(* CODESYS project SPT_Utilities.library
   Version: 4.0.1
   Title: SPT Utilities
   DefaultNamespace: SPT_Utilities
   Placeholder: SPT Utilities
   Company: Beckhoff Automation LLC

Project tree, tasks and I/O mapping:
  libraries: SPT Base Types, * (Beckhoff Automation LLC); SPT Event Logger, * (Beckhoff Automation LLC); Tc2_Standard, * (Beckhoff Automation GmbH); Tc2_System, * (Beckhoff Automation GmbH); Tc3_EventLogger, * (Beckhoff Automation GmbH); Tc3_JsonXml, * (Beckhoff Automation GmbH); Tc3_Module, * (Beckhoff Automation GmbH)
  Analog Scaling/
    DUT/
      data type ST_ScalingParameters
    function F_ApplyScaling [ST]
  Buffers/
    Array ANY Datatype/
      function block FB_ArrayAny [ST]: CheckBoundary, Delete, Enable, Exchange, Insert, LowerBoundary, Reset, UpperBoundary
    Buffers ANY Datatype/
      function block FB_AnyBase [ST]: CheckBoundary, CheckDataSize, CheckPointer, ClearError, Empty, Enable, Full, LowerBoundary, UpperBoundary
      function block FB_BufferAny [ST]: Push, Reset
      function block FB_FIFOAny [ST]: Pop, Push, Reset
      function block FB_LIFOAny [ST]: Pop, Push, Reset
      function block FB_RingAny [ST]: Pop, Push, Reset
      function IncrementBy1ToLimit [ST]
    function block FB_FIFO_ULINT_Array [ST]: AddEntry, EntryCount, LastInValue, NextOutValue, RemoveEntry
  File Handlers/
    function block FB_Component_JsonFileHandler [ST]: GetDataTypeFromPVOID, CreateEvents, Monitoring, CyclicLogic, ClearDocument, LoadFile, ReadAny, ReadBool, ReadDInt, ReadLREAL, ReadString, ReadSymbol, Reset, UpdateAny, UpdateBool, UpdateDInt, UpdateLREAL, UpdateString, UpdateSymbol, LoadFileSequence, SaveFileSequence, Path, Timeout
    interface I_FileHandler: ClearDocument, LoadFile, ReadBool, ReadDInt, ReadLREAL, ReadString, ReadSymbol, Reset, Timeout, UpdateAny, UpdateBool, UpdateDInt, UpdateLREAL, UpdateString, UpdateSymbol
  Helper/
    function F_CompareLREAL [ST]
    function F_CompareREAL [ST]
    function F_LREAL_RoundToPlace [ST]
    function block FB_SimpleRateLimiter [ST]
  Project Information/
    function F_GetCompany [ST]
    function F_GetTitle [ST]
    function F_GetVersion [ST]
  String Helper/
    function block FB_StringHelper [ST]: GetExtensionOrVarName, GetFileNameFromPath, GetFilePath, GetName, GetPath, GetSymbolPath, RemoveFirstChar, RemoveLastChar, StringToCharArray, ValidInput
  Trace Listener/
    function block FB_MessageListener [ST]: Listener, OnMessageSent
    function block FB_TraceListenerBase [ST]: CyclicLogic, Initialize, OnTraceReceived
    interface I_TraceListener: OnTraceReceived
    data type ST_TraceMessage
  Tree_IndexBased/
    function block FB_Tree_IndexBased [ST]: AddNodeAsChildByName, GetIndexByName, Initialize
    interface I_Tree_IndexBased: AddNodeAsChildByName
    data type ST_Tree_IndexBased_Node
  Version/
    global variables Global_Version
  00000000-0000-0000-0000-000000000000|LICENSE
  LICENSE
  global variables Parameter_Utilities
*)

// Analog Scaling/DUT/ST_ScalingParameters
TYPE ST_ScalingParameters :
	STRUCT
		Input_Minimum  : LREAL := 0;
		Input_Maximum  : LREAL := 100;
		Output_Minimum : LREAL := 0;
		Output_Maximum : LREAL := 4096;
	END_STRUCT
END_TYPE

// Trace Listener/ST_TraceMessage
TYPE ST_TraceMessage :
	STRUCT
		Timestamp : T_MaxString;
		Source	  : T_MaxString;
		Context	  : T_MaxString;
		ScanCount : UDINT;
		Flags	  : UDINT;
		Message	  : T_MaxString;
		Json	  : T_MaxString;
	END_STRUCT
END_TYPE

// Tree_IndexBased/ST_Tree_IndexBased_Node
TYPE ST_Tree_IndexBased_Node :
	STRUCT
		Name	   : STRING;
		ChildCount : DINT;
		Parent	   : DINT;
		Children   : ARRAY[0..15] OF DINT;
		Depth	   : DINT;
	END_STRUCT
END_TYPE

// Version/Global_Version
{attribute 'TcGenerated'}
{attribute 'no-analysis'}
{attribute 'linkalways'}
// This function has been automatically generated from the project information.
VAR_GLOBAL CONSTANT
	{attribute 'const_non_replaced'}
	stLibVersion_SPT_Utilities : ST_LibVersion := (iMajor := 4, iMinor := 0, iBuild := 1, iRevision := 0, nFlags := 1, sVersion := '4.0.1');
END_VAR

// Parameter_Utilities
{attribute 'qualified_only'}
VAR_GLOBAL CONSTANT
	FILE_SIZE : UDINT := 1300000; // Number of Characters in file to read via Read/Write Symbol
END_VAR

// Analog Scaling/F_ApplyScaling
FUNCTION F_ApplyScaling : LREAL
VAR_INPUT
	X		   : LREAL;
	Parameters : ST_ScalingParameters;
END_VAR

VAR
	Slope : LREAL;
END_VAR

IF Parameters.Input_Minimum >= Parameters.Input_Maximum THEN
	// Error -- no span to scale
	F_ApplyScaling := 0;
	RETURN;
ELSIF Parameters.Output_Minimum >= Parameters.Output_Maximum THEN
	// Error -- no span to scale
	F_ApplyScaling := 0;
	RETURN;
END_IF

// Input is pegged
IF X <= Parameters.Input_Minimum THEN
	F_ApplyScaling := Parameters.Output_Minimum;
	RETURN;
ELSIF X >= Parameters.Input_Maximum THEN
	F_ApplyScaling := Parameters.Output_Maximum;
	RETURN;
END_IF

// I/O ok--scale it
IF (Parameters.Input_Maximum - Parameters.Input_Minimum) <> 0.0 THEN
	Slope := (Parameters.Output_Maximum - Parameters.Output_Minimum) / (Parameters.Input_Maximum - Parameters.Input_Minimum);
ELSE
	Slope := 0.0;
END_IF

F_ApplyScaling := Slope * (X - Parameters.Input_Minimum) + Parameters.Output_Minimum;

END_FUNCTION

// Buffers/Array ANY Datatype/FB_ArrayAny
(*
	Manipulation of an any array
	ELEMENTS AT _locATIONS CAN BE ADDED, REMOVED or EXCHANGED
	THE FUNCTION B_locK DOES NOT CARE ABOUT FULL OR 
	VARIABLE SIZED 
	ANY 
	array *)

//  !!! Use the dereferenced buffer (^) in CASE OF [*] defined arrays inside an FB !!!
FUNCTION_BLOCK FB_ArrayAny EXTENDS FB_BaseFB
VAR
	// Properties
	_LowerBoundary : DINT;
	_UpperBoundary : DINT;
	_Enable		   : BOOL := TRUE;

	// Internal variables
	_Location : DINT;
END_VAR

METHOD PRIVATE CheckBoundary : BOOL
VAR_INPUT
END_VAR
CheckBoundary := TRUE;
IF (_LowerBoundary >= _UpperBoundary) OR (_LowerBoundary < 0) THEN
	IF NOT _Error THEN // avoid retrigger
		Trace(CONCAT(InstancePath, ': Boundary sizes incorrect (L>=U) OR (L<0)'));
	END_IF

	_Error		  := TRUE;
	CheckBoundary := FALSE;
END_IF
END_METHOD

METHOD Delete : BOOL
VAR_INPUT
	ArrayIn	 : ANY;
	DataIn	 : ANY;
	Location : DINT;
END_VAR
Delete := FALSE;
IF ArrayIn.pValue = 0 THEN
	IF NOT _Error THEN
		Trace(CONCAT(InstancePath, ': Missing ANY input when calling ARRAY'));
		_Error := TRUE;
		RETURN;
	END_IF
END_IF

IF NOT CheckBoundary() THEN
	RETURN;
END_IF

_Location := Location - _LowerBoundary;
IF _Enable THEN
	IF Location <= _UpperBoundary AND Location >= _LowerBoundary THEN
		MEMMOVE(ADR(ArrayIn.pValue[DataIn.diSize * _Location]), ADR(ArrayIn.pValue[DataIn.diSize * (_Location + 1)]), TO_UDINT((_UpperBoundary - Location) * DataIn.diSize));
		MEMSET(ADR(ArrayIn.pValue[(_UpperBoundary - _LowerBoundary) * DataIn.diSize]), 0, TO_UDINT(DataIn.diSize)); // last _location clear
	ELSE
		Trace('Attempt to remove from invalid _location in ARRAY');
	END_IF
END_IF
END_METHOD

PROPERTY Enable : BOOL
SET
_Enable := Enable;
END_SET
END_PROPERTY

METHOD Exchange : BOOL
VAR_INPUT
	ArrayIn	 : ANY;
	DataIn	 : ANY;
	Location : DINT;
END_VAR
Exchange := FALSE;
IF ArrayIn.pValue = 0 THEN
	IF NOT _Error THEN
		Trace(CONCAT(InstancePath, ': Missing ANY input when calling ARRAY'));
		_Error := TRUE;
		RETURN;
	END_IF
END_IF

IF NOT CheckBoundary() THEN
	RETURN;
END_IF

_Location := Location - _LowerBoundary;
IF Location <= _UpperBoundary AND location >= _LowerBoundary THEN
	memcpy(ADR(ArrayIn.pValue[_Location * DataIn.diSize]), DataIn.pValue, TO_UDINT(DataIn.diSize)); // insert new data on _location
	Exchange := TRUE;
ELSE
	Trace('Attempt to exchange at invalid _location in ARRAY');
END_IF
END_METHOD

METHOD Insert : BOOL
VAR_INPUT
	ArrayIn	 : ANY;
	DataIn	 : ANY;
	Location : DINT;
END_VAR
Insert := FALSE;
IF DataIn.pValue = 0 OR_ELSE ArrayIn.pValue = 0 THEN
	IF NOT _Error THEN
		Trace(CONCAT(InstancePath, ': Missing ANY input when calling ARRAY'));
		_Error := TRUE;
		RETURN;
	END_IF
END_IF

IF NOT CheckBoundary() THEN
	RETURN;
END_IF

_Location := Location - _LowerBoundary;
IF Location >= _LowerBoundary THEN
	IF Location < _UpperBoundary THEN
		MEMMOVE(ADR(ArrayIn.pValue[DataIn.diSize * (_Location + 1)]), ADR(ArrayIn.pValue[DataIn.diSize * _Location]), TO_UDINT((_UpperBoundary - Location) * DataIn.diSize));
	END_IF

	memcpy(ADR(ArrayIn.pValue[_Location * DataIn.diSize]), DataIn.pValue, TO_UDINT(DataIn.diSize)); // insert new data on _location
ELSE
	Trace('Attempt to insert at invalid _location in ARRAY');
END_IF
END_METHOD

PROPERTY LowerBoundary : DINT
SET
_LowerBoundary := LowerBoundary;
END_SET
END_PROPERTY

METHOD Reset
VAR_INPUT
	ArrayIn : ANY;
END_VAR
IF ArrayIn.pValue = 0 THEN
	IF NOT _Error THEN
		Trace(CONCAT(InstancePath, ': Missing ANY input when calling ARRAY'));
		_Error := TRUE;
		RETURN;
	END_IF
END_IF

IF NOT CheckBoundary() THEN
	RETURN;
END_IF

MEMSET(ArrayIn.pValue, 0, TO_UDINT(ArrayIn.diSize));
END_METHOD

PROPERTY UpperBoundary : DINT
SET
_UpperBoundary := UpperBoundary;
END_SET
END_PROPERTY

END_FUNCTION_BLOCK

// Buffers/Buffers ANY Datatype/FB_AnyBase
(*
	Any Base extends from FB_BaseFB to get Tracing and _Error
	This houses the boundaries, Enable, Full/Empty properties 
	that all the buffer types have.
*)
FUNCTION_BLOCK FB_AnyBase EXTENDS FB_BaseFB
VAR
	// Properties
	_LowerBoundary : DINT;
	_UpperBoundary : DINT;
	_Enable		   : BOOL;
	_Empty		   : BOOL := TRUE;
	_Full		   : BOOL := FALSE;
END_VAR

METHOD PROTECTED CheckBoundary : BOOL
VAR_INPUT
END_VAR
CheckBoundary := TRUE;
IF (_LowerBoundary >= _UpperBoundary) OR (_LowerBoundary < 0) THEN
	IF NOT _Error THEN // avoid retrigger
		Trace('Boundary sizes incorrect (L>=U) OR (L<0)');
	END_IF

	_Error		  := TRUE;
	CheckBoundary := FALSE;
END_IF
END_METHOD

METHOD CheckDataSize : BOOL
VAR_INPUT
	BufferIn : ANY; // Entire Buffer Array to be cleared
	DataIn	 : ANY; // Single array index for size calculation
END_VAR
CheckDataSize := TRUE;
IF BufferIn.diSize <> (_UpperBoundary - _LowerBoundary + 1) * DataIn.diSize THEN
	IF NOT _Error THEN // avoid retrigger
		Trace(CONCAT(InstancePath, ': Data sizes do not match.'));
	END_IF

	_Error		  := TRUE;
	CheckDataSize := FALSE;
END_IF
END_METHOD

METHOD CheckPointer : BOOL
VAR_INPUT
	pValue : POINTER TO BYTE;
END_VAR
CheckPointer := TRUE;
IF pValue = 0 THEN
	IF NOT _Error THEN
		Trace(CONCAT(InstancePath, ': Missing pointer input when calling.'));
	END_IF

	_Error		 := TRUE;
	CheckPointer := FALSE;
END_IF
END_METHOD

METHOD ClearError
VAR_INPUT
	MethodName : STRING;
END_VAR

VAR
	msg : STRING;
END_VAR
_Error := FALSE;
msg	   := CONCAT(InstancePath, ': Error cleared during ');
msg	   := CONCAT(msg, MethodName);
TRACE(msg);
END_METHOD

PROPERTY Empty : BOOL
GET
Empty := _Empty;
END_GET
END_PROPERTY

PROPERTY Enable : BOOL
GET
Enable := _Enable;
END_GET
SET
_Enable := Enable;
END_SET
END_PROPERTY

PROPERTY Full : BOOL
GET
Full := _Full;
END_GET
END_PROPERTY

PROPERTY LowerBoundary : DINT
SET
_LowerBoundary := LowerBoundary;
END_SET
END_PROPERTY

PROPERTY UpperBoundary : DINT
SET
_UpperBoundary := UpperBoundary;
END_SET
END_PROPERTY

END_FUNCTION_BLOCK

// Buffers/Buffers ANY Datatype/FB_BufferAny
(*
	simple memory buffer
	WHEN FULL NO MORE ELEMENTS CAN BE ADDED
	VARIABLE SIZED 
	ANY 
	array *)

//  !!! Use the dereferenced buffer (^) in CASE OF [*] defined arrays inside an FB !!!
FUNCTION_BLOCK FB_BufferAny EXTENDS FB_AnyBase
VAR
	// Internal Variables
	BufferIndex : DINT := 0; // write pointer in buffer
END_VAR

METHOD Push : BOOL
VAR_INPUT
	BufferIn : ANY; // Entire Buffer Array to be cleared
	DataIn	 : ANY; // Single array index for size calculation
END_VAR

VAR
	_TotalSlots : DINT;
END_VAR
IF _Error THEN
	ClearError('Push');
END_IF

IF NOT CheckPointer(pValue := BufferIn.pValue) THEN
	RETURN;
END_IF

IF NOT CheckPointer(pValue := DataIn.pValue) THEN
	RETURN;
END_IF

IF NOT CheckBoundary() THEN
	RETURN;
END_IF

IF _Enable THEN
	IF _Full THEN
		_Error := TRUE;
		Trace('Attempt to write to full buffer');
	ELSE
		// Push DataIn to BufferIn at Index
		memcpy(ADR(BufferIn.pValue[TO_DINT(BufferIndex) * DataIn.diSize]), DataIn.pValue, TO_UDINT(DataIn.diSize));

		//		
		_TotalSlots := _UpperBoundary - _LowerBoundary + 1;

		// Increment buffer index
		BufferIndex := BufferIndex + 1;

		//
		_Full  := BufferIndex = _TotalSlots;
		_Empty := FALSE;
	END_IF
END_IF
END_METHOD

METHOD Reset
VAR_INPUT
	BufferIn : ANY; // Entire Buffer Array to be cleared
	DataIn	 : ANY; // Single array index for size calculation
END_VAR

VAR
	_TotalSlots : DINT;
END_VAR
IF _Error THEN
	ClearError('Reset');
END_IF

IF NOT CheckPointer(pValue := BufferIn.pValue) THEN
	RETURN;
END_IF

IF NOT CheckPointer(pValue := DataIn.pValue) THEN
	RETURN;
END_IF

IF NOT CheckBoundary() THEN
	RETURN;
END_IF

// Check Data Size mismatch
IF NOT CheckDataSize(BufferIn := BufferIn, DataIn := DataIn) THEN
	RETURN;
END_IF

//		
_TotalSlots := _UpperBoundary - _LowerBoundary + 1;

//
BufferIndex := 0;
_Full		:= FALSE;
_Empty		:= TRUE;
memset(BufferIn.pValue, 0, TO_UDINT(_TotalSlots * DataIn.diSize)); // get element size
_Error := FALSE;
END_METHOD

END_FUNCTION_BLOCK

// Buffers/Buffers ANY Datatype/FB_FIFOAny
(*
	FIFO circular (RING) memory buffer, loops around the available buffer
	MOST EFFICIENT FIFO, avoids unnecessary copying in the buffer
	WHEN FULL NO MORE ELEMENTS CAN BE ADDED
	VARIABLE SIZED 
	ANY 
	array *)

//  !!! Use the dereferenced buffer (^) in CASE OF [*] defined arrays inside an FB !!!
FUNCTION_BLOCK FB_FIFOAny EXTENDS FB_AnyBase
VAR
	// Internal Variables
	ReadBufferIndex	 : DINT := 0; // read pointer in buffer, Tail
	WriteBufferIndex : DINT := 0; // write pointer in buffer, Head
END_VAR

METHOD Pop : BOOL
VAR_INPUT
	FIFOIn	: ANY; // Entire FIFO Array
	DataOut : ANY; // Single Array Index of data to push
END_VAR

VAR
	_TotalSlots : DINT;
END_VAR
IF _Error THEN
	ClearError('Pop');
END_IF

IF NOT CheckPointer(pValue := FIFOIn.pValue) THEN
	RETURN;
END_IF

IF NOT CheckPointer(pValue := DataOut.pValue) THEN
	RETURN;
END_IF

IF NOT CheckBoundary() THEN
	RETURN;
END_IF

IF EMPTY THEN
	_Error := TRUE;
	Trace('Attempt to read from empty Fifo buffer');
ELSE
	// Clear memory in DataOut
	memset(DataOut.pValue, 0, TO_UDINT(DataOut.diSize));

	// Pop FIFO at Index to DataOut
	memcpy(DataOut.pValue, ADR(FIFOIn.pValue[(ReadBufferIndex) * DataOut.diSize]), TO_UDINT(DataOut.diSize));

	// Clear memory in FIFO at Index
	memset(ADR(FIFOIn.pValue[(ReadBufferIndex) * DataOut.diSize]), 0, TO_UDINT(DataOut.diSize));

	//		
	_TotalSlots := _UpperBoundary - _LowerBoundary + 1;

	// Increment buffer index or reset to 0
	ReadBufferIndex := IncrementBy1ToLimit(ReadBufferIndex, _TotalSlots);

	// Determine if Buffer is empty
	IF (WriteBufferIndex = ReadBufferIndex) THEN
		_Empty := TRUE;
	ELSE
		_Empty := FALSE;
	END_IF

	_Full := FALSE;
END_IF
END_METHOD

METHOD Push : BOOL
VAR_INPUT
	FIFOIn : ANY; // Entire FIFO Array
	DataIn : ANY; // Single Array Index of data to push
END_VAR

VAR
	_UsedSlots	: DINT;
	_TotalSlots : DINT;
END_VAR
IF _Error THEN
	ClearError('Push');
END_IF

IF NOT CheckPointer(pValue := FIFOIn.pValue) THEN
	RETURN;
END_IF

IF NOT CheckPointer(pValue := DataIn.pValue) THEN
	RETURN;
END_IF

IF NOT CheckBoundary() THEN
	RETURN;
END_IF

IF _Enable THEN
	IF _Full THEN
		_Error := TRUE;
		Trace('Attempt to write to full buffer');
	ELSE
		// Push DataIn to FIFO at Index
		memcpy(ADR(FIFOIn.pValue[(WriteBufferIndex) * DataIn.diSize]), DataIn.pValue, TO_UDINT(DataIn.diSize));

		//		
		_TotalSlots := _UpperBoundary - _LowerBoundary + 1;

		// Increment buffer index or reset to 0
		WriteBufferIndex := IncrementBy1ToLimit(WriteBufferIndex, _TotalSlots);

		// Calc Used Buffer Size
		IF (WriteBufferIndex > ReadBufferIndex) THEN
			_UsedSlots := WriteBufferIndex - ReadBufferIndex;
		ELSIF WriteBufferIndex < ReadBufferIndex THEN
			_UsedSlots := (WriteBufferIndex + _TotalSlots) - ReadBufferIndex;
		END_IF

		// Determine if Buffer is full
		IF WriteBufferIndex = ReadBufferIndex THEN
			_Full := TRUE;
		ELSIF _UsedSlots = _TotalSlots THEN
			_Full := TRUE;
		ELSE
			_Full := FALSE;
		END_IF

		_Empty := FALSE;
	END_IF
END_IF
END_METHOD

METHOD Reset : BOOL
VAR_INPUT
	FIFOIn	: ANY; // Entire FIFO Array
	DataIn	: ANY; // Single Array Index for size calculation
	DataOut : ANY; // Entire Data Out Array
END_VAR

VAR
	_TotalSlots : DINT;
END_VAR
IF _Error THEN
	ClearError('Reset');
END_IF

IF NOT CheckPointer(pValue := FIFOIn.pValue) THEN
	RETURN;
END_IF

IF NOT CheckPointer(pValue := DataIn.pValue) THEN
	RETURN;
END_IF

IF NOT CheckPointer(pValue := DataOut.pValue) THEN
	RETURN;
END_IF

IF NOT CheckBoundary() THEN
	RETURN;
END_IF

// Check Data Size mismatch
IF NOT CheckDataSize(BufferIn := FIFOIn, DataIn := DataIn) THEN
	RETURN;
END_IF

//		
_TotalSlots := _UpperBoundary - _LowerBoundary + 1;

//
WriteBufferIndex := ReadBufferIndex := 0;
_Full								:= FALSE;
_Empty								:= TRUE;
memset(DataOut.pValue, 0, TO_UDINT(DataOut.diSize));
memset(FIFOIn.pValue, 0, TO_UDINT(_TotalSlots * DataIn.diSize)); // get element size
_Error := FALSE;
END_METHOD

END_FUNCTION_BLOCK

// Buffers/Buffers ANY Datatype/IncrementBy1ToLimit
FUNCTION IncrementBy1ToLimit : DINT
VAR_INPUT
	In		   : DINT;
	UpperLimit : DINT;
END_VAR

IncrementBy1ToLimit := In + 1;
IF IncrementBy1ToLimit >= UpperLimit THEN
	IncrementBy1ToLimit := 0; // Begining of memory for the buffer
END_IF

END_FUNCTION

// Buffers/Buffers ANY Datatype/FB_LIFOAny
(*
	LIFO (STACK) memory
	WHEN FULL NO MORE ELEMENTS CAN BE ADDED
	VARIABLE SIZED 
	ANY 
	array *)

//  !!! Use the dereferenced buffer (^) in CASE OF [*] defined arrays inside an FB !!!
FUNCTION_BLOCK FB_LIFOAny EXTENDS FB_AnyBase
VAR
	// Internal Variables
	LifoIndex : DINT := 0; // Index to LIFO
END_VAR

METHOD Pop : BOOL
VAR_INPUT
	LIFOIn	: ANY; // Entire LIFO Array
	DataOut : ANY; // Single Array Index of data to pop
END_VAR
IF _Error THEN
	ClearError('Pop');
END_IF

IF NOT CheckPointer(pValue := LIFOIn.pValue) THEN
	RETURN;
END_IF

IF NOT CheckPointer(pValue := DataOut.pValue) THEN
	RETURN;
END_IF

IF NOT CheckBoundary() THEN
	RETURN;
END_IF

IF EMPTY THEN
	_Error := TRUE;
	Trace('Attempt to read from empty LIFO buffer');
ELSE
	// Reset output
	memset(DataOut.pValue, 0, TO_UDINT(DataOut.diSize));
	LifoIndex := LifoIndex - 1;
	memcpy(DataOut.pValue, ADR(LIFOIn.pValue[LifoIndex * DataOut.diSize]), TO_UDINT(DataOut.diSize));
	memset(ADR(LIFOIn.pValue[LifoIndex * DataOut.diSize]), 0, TO_UDINT(DataOut.diSize));
	_Empty := LifoIndex = 0;
	_Full  := FALSE;
END_IF
END_METHOD

METHOD Push : BOOL
VAR_INPUT
	LIFOIn : ANY; // Entire LIFO Array
	DataIn : ANY; // Single Array Index of data to push
END_VAR

VAR
	_TotalSlots : DINT;
END_VAR
IF _Error THEN
	ClearError('Push');
END_IF

IF NOT CheckPointer(pValue := LIFOIn.pValue) THEN
	RETURN;
END_IF

IF NOT CheckPointer(pValue := DataIn.pValue) THEN
	RETURN;
END_IF

IF NOT CheckBoundary() THEN
	RETURN;
END_IF

IF _Enable THEN
	IF _Full THEN
		_Error := TRUE;
		Trace('Attempt to write to full LIFO');
	ELSE
		// Push DataIn to BufferIn at Index
		memcpy(ADR(LIFOIn.pValue[LifoIndex * DataIn.diSize]), DataIn.pValue, TO_UDINT(DataIn.diSize));

		//		
		_TotalSlots := _UpperBoundary - _LowerBoundary + 1;

		// Increment buffer index
		LifoIndex := LifoIndex + 1;

		//
		_Full  := LifoIndex = _TotalSlots;
		_Empty := FALSE;
	END_IF
END_IF
END_METHOD

METHOD Reset
VAR_INPUT
	LIFOIn	: ANY;
	DataIn	: ANY;
	DataOut : ANY;
END_VAR

VAR
	_TotalSlots : DINT;
END_VAR
IF _Error THEN
	ClearError('Reset');
END_IF

IF NOT CheckPointer(pValue := LIFOIn.pValue) THEN
	RETURN;
END_IF

IF NOT CheckPointer(pValue := DataIn.pValue) THEN
	RETURN;
END_IF

IF NOT CheckPointer(pValue := DataOut.pValue) THEN
	RETURN;
END_IF

IF NOT CheckBoundary() THEN
	RETURN;
END_IF

// Check Data Size mismatch
IF NOT CheckDataSize(BufferIn := LIFOIn, DataIn := DataIn) THEN
	RETURN;
END_IF

//		
_TotalSlots := _UpperBoundary - _LowerBoundary + 1;

//
LifoIndex := 0;
_Full	  := FALSE;
_Empty	  := TRUE;
memset(DataOut.pValue, 0, TO_UDINT(DataOut.diSize));
memset(LIFOIn.pValue, 0, TO_UDINT(_TotalSlots * DataIn.diSize)); // get element size
_Error := FALSE;
END_METHOD

END_FUNCTION_BLOCK

// Buffers/Buffers ANY Datatype/FB_RingAny
(*
	Ring circular memory buffer, loops around the available buffer
	MOST EFFICIENT ring, avoids unnecessary copying in the buffer
	WHEN FULL THE NEW ELEMENT IS ADDED AND THE FIRST/NEXT ELEMENT IS LOST
	VARIABLE SIZED 
	ANY 
	array 
*)

//  !!! Use the dereferenced buffer (^) in CASE OF [*] defined arrays inside an FB !!!
FUNCTION_BLOCK FB_RingAny EXTENDS FB_AnyBase
VAR
	// Internal Variables
	ReadBufferIndex	 : DINT := 0; // read pointer in buffer, Tail
	WriteBufferIndex : DINT := 0; // write pointer in buffer, Head
END_VAR

METHOD Pop : BOOL
VAR_INPUT
	RingIn	: ANY; // Entire Ring Array
	DataOut : ANY; // Single Array Index of data to push
END_VAR

VAR
	_TotalSlots : DINT;
END_VAR
IF _Error THEN
	ClearError('Pop');
END_IF

IF NOT CheckPointer(pValue := RingIn.pValue) THEN
	RETURN;
END_IF

IF NOT CheckPointer(pValue := DataOut.pValue) THEN
	RETURN;
END_IF

IF NOT CheckBoundary() THEN
	RETURN;
END_IF

IF EMPTY THEN
	_Error := TRUE;
	Trace('Attempt to read from empty Ring buffer');
ELSE
	// Clear memory at DataOut
	memset(DataOut.pValue, 0, TO_UDINT(DataOut.diSize));

	// Pop Ring at Index to DataOut
	memcpy(DataOut.pValue, ADR(RingIn.pValue[TO_DINT(ReadBufferIndex) * DataOut.diSize]), TO_UDINT(DataOut.diSize));

	// CLear memory in Ring at Index
	memset(ADR(RingIn.pValue[TO_DINT(ReadBufferIndex) * DataOut.diSize]), 0, TO_UDINT(DataOut.diSize));

	//		
	_TotalSlots := _UpperBoundary - _LowerBoundary + 1;

	// Increment buffer index or reset to 0
	ReadBufferIndex := IncrementBy1ToLimit(ReadBufferIndex, _TotalSlots);

	// Determine if Buffer is empty
	IF (WriteBufferIndex = ReadBufferIndex) THEN
		_Empty := TRUE;
	ELSE
		_Empty := FALSE;
	END_IF

	_Full := FALSE;
END_IF
END_METHOD

METHOD Push : BOOL
VAR_INPUT
	RingIn : ANY; // Entire Ring Array
	DataIn : ANY; // Single Array Index of data to push
END_VAR

VAR
	_UsedSlots	: DINT;
	_TotalSlots : DINT;
END_VAR
IF _Error THEN
	ClearError('Push');
END_IF

IF NOT CheckPointer(pValue := RingIn.pValue) THEN
	RETURN;
END_IF

IF NOT CheckPointer(pValue := DataIn.pValue) THEN
	RETURN;
END_IF

IF NOT CheckBoundary() THEN
	RETURN;
END_IF

IF _Enable THEN
	// Push DataIn to next location in Ring
	memcpy(ADR(RingIn.pValue[TO_DINT(WriteBufferIndex) * DataIn.diSize]), DataIn.pValue, TO_UDINT(DataIn.diSize));

	//		
	_TotalSlots := _UpperBoundary - _LowerBoundary + 1;

	// Increment buffer index or reset to 0
	WriteBufferIndex := IncrementBy1ToLimit(WriteBufferIndex, _TotalSlots);

	// Calc Used Buffer Size
	IF (WriteBufferIndex > ReadBufferIndex) THEN
		_UsedSlots := WriteBufferIndex - ReadBufferIndex;
	ELSIF WriteBufferIndex < ReadBufferIndex THEN
		_UsedSlots := (WriteBufferIndex + _TotalSlots) - ReadBufferIndex;
	END_IF

	// Determine if Buffer is full
	IF WriteBufferIndex = ReadBufferIndex THEN
		_Full := TRUE;
	ELSIF _UsedSlots = _TotalSlots THEN
		_Full := TRUE;
	ELSE
		_Full := FALSE;
	END_IF

	_Empty := FALSE;
END_IF
END_METHOD

METHOD Reset
VAR_INPUT
	RingIn	: ANY; // Entire Ring Array
	DataIn	: ANY; // Single Array Index for size calculation
	DataOut : ANY; // Entire Data Out Array
END_VAR

VAR
	_TotalSlots : DINT;
END_VAR
IF _Error THEN
	ClearError('Reset');
END_IF

IF NOT CheckPointer(pValue := RingIn.pValue) THEN
	RETURN;
END_IF

IF NOT CheckPointer(pValue := DataIn.pValue) THEN
	RETURN;
END_IF

IF NOT CheckPointer(pValue := DataOut.pValue) THEN
	RETURN;
END_IF

IF NOT CheckBoundary() THEN
	RETURN;
END_IF

// Check Data Size mismatch
IF NOT CheckDataSize(BufferIn := RingIn, DataIn := DataIn) THEN
	RETURN;
END_IF

//		
_TotalSlots := _UpperBoundary - _LowerBoundary + 1;

//
WriteBufferIndex := ReadBufferIndex := 0;
_Full								:= FALSE;
_Empty								:= TRUE;
memset(DataOut.pValue, 0, TO_UDINT(DataOut.diSize));
memset(RingIn.pValue, 0, TO_UDINT(_TotalSlots * DataIn.diSize)); // get element size
_Error := FALSE;
END_METHOD

END_FUNCTION_BLOCK

// Buffers/FB_FIFO_ULINT_Array
// A general purpose FIFO buffer for the ULINT (64-bit Unsigned Integer) datatype
FUNCTION_BLOCK FB_FIFO_ULINT_Array
VAR_IN_OUT
	Buffer : ARRAY[*] OF ULINT;
END_VAR

VAR
	_EntryCount : DINT;
END_VAR

// Adds an entry to the buffer
METHOD AddEntry : BOOL // TRUE if entry was accepted, FALSE if buffer is full
VAR_INPUT
	Entry : ULINT; // Entry to add
END_VAR

VAR
	i : DINT;
END_VAR
IF (LOWER_BOUND(Buffer, 1) + _EntryCount - 1) > UPPER_BOUND(Buffer, 1) THEN
	AddEntry := FALSE; // FIFO is full
ELSE
	FOR i := UPPER_BOUND(Buffer, 1) - 1 TO LOWER_BOUND(Buffer, 1) BY -1 DO
		Buffer[i + 1] := Buffer[i];
	END_FOR

	Buffer[LOWER_BOUND(Buffer, 1)] := Entry;
	_EntryCount					   := _EntryCount + 1;
	AddEntry					   := TRUE;
END_IF
END_METHOD

// Returns the number of entries in the buffer
PROPERTY EntryCount : DINT
GET
EntryCount := _EntryCount;
END_GET
END_PROPERTY

// Returns the last entry placed in the buffer
PROPERTY LastInValue : ULINT
GET
IF _EntryCount = 0 THEN
	LastInValue := 0;
ELSE
	LastInValue := Buffer[LOWER_BOUND(Buffer, 1)];
END_IF
END_GET
END_PROPERTY

// Returns the head entry of the buffer
PROPERTY NextOutValue : ULINT
GET
IF _EntryCount = 0 THEN
	NextOutValue := 0;
ELSE
	NextOutValue := Buffer[LOWER_BOUND(Buffer, 1) + _EntryCount - 1];
END_IF
END_GET
END_PROPERTY

// Removes head entry from the buffer
METHOD RemoveEntry : BOOL // TRUE if entry was removed, FALSE if the buffer was already empty
VAR
	i : DINT;
END_VAR
IF _EntryCount = 0 THEN
	RemoveEntry := FALSE;
ELSE
	IF (LOWER_BOUND(Buffer, 1) + _EntryCount - 1) <= UPPER_BOUND(Buffer, 1) THEN
		Buffer[LOWER_BOUND(Buffer, 1) + _EntryCount - 1] := 0;
		_EntryCount										 := _EntryCount - 1;
		RemoveEntry										 := TRUE;
	END_IF
END_IF
END_METHOD

END_FUNCTION_BLOCK

// File Handlers/FB_Component_JsonFileHandler
FUNCTION_BLOCK FB_Component_JsonFileHandler EXTENDS FB_ComponentBase IMPLEMENTS I_FileHandler
VAR
	_Path : STRING;

	// Json Management 
	FileRead			  : BOOL;
	FileSave			  : BOOL;
	FileLoadOk			  : BOOL;
	FileSaveOk			  : BOOL;
	JsonFileMachineConfig : FB_JsonDomParser;
	JsonDoc				  : SJsonValue;
	JsonProp			  : SJsonValue;
	JsonRW_DataType		  : FB_JsonReadWriteDatatype;
	i					  : UDINT;
	SeqLoad				  : UDINT;
	SeqSave				  : UDINT;
	TonTimeout			  : TON;
	_Timeout			  : TIME := T#1S;
	LoadDone			  : BOOL;

	// Folder Management
	fbCreateDir : FB_CreateDir;
	strHelp		: FB_StringHelper;

	// Symbol
	JsonReadWriteDataType : FB_JsonREadWriteDatatype;
	ValueJson			  : STRING(Parameter_Utilities.FILE_SIZE);
	hr					  : HRESULT;

	// Alarms
	JsonFileHandlerAlarms : ARRAY[1..JSON_FILE_ALARM_COUNT] OF FB_TcAlarm;
END_VAR

VAR CONSTANT
	JSON_FILE_ALARM_COUNT : UDINT := 3;
END_VAR

METHOD GetDataTypeFromPVOID : STRING
VAR_INPUT
	pData : pvoid; // address of symbol
END_VAR

VAR
	nData	   : UDINT;
	resultSize : ARRAY[0..256] OF STRING;
END_VAR
nData := SIZEOF(pData);
IF JsonRW_DataType.GetDatatypeNameByAddress(SIZEOF(BOOL), pData) = 'BOOL' THEN
	GetDataTypeFromPVOID := 'BOOL';
	RETURN;
END_IF

IF JsonRW_DataType.GetDatatypeNameByAddress(SIZEOF(BYTE), pData) = 'BYTE' THEN
	GetDataTypeFromPVOID := 'BYTE';
	RETURN;
END_IF

IF JsonRW_DataType.GetDatatypeNameByAddress(SIZEOF(WORD), pData) = 'WORD' THEN
	GetDataTypeFromPVOID := 'WORD';
	RETURN;
END_IF

IF JsonRW_DataType.GetDatatypeNameByAddress(SIZEOF(DWORD), pData) = 'DWORD' THEN
	GetDataTypeFromPVOID := 'DWORD';
	RETURN;
END_IF

IF JsonRW_DataType.GetDatatypeNameByAddress(SIZEOF(SINT), pData) = 'SINT' THEN
	GetDataTypeFromPVOID := 'SINT';
	RETURN;
END_IF

IF JsonRW_DataType.GetDatatypeNameByAddress(SIZEOF(USINT), pData) = 'USINT' THEN
	GetDataTypeFromPVOID := 'USINT';
	RETURN;
END_IF

IF JsonRW_DataType.GetDatatypeNameByAddress(SIZEOF(INT), pData) = 'INT' THEN
	GetDataTypeFromPVOID := 'INT';
	RETURN;
END_IF

IF JsonRW_DataType.GetDatatypeNameByAddress(SIZEOF(UINT), pData) = 'UINT' THEN
	GetDataTypeFromPVOID := 'UINT';
	RETURN;
END_IF

IF JsonRW_DataType.GetDatatypeNameByAddress(SIZEOF(DINT), pData) = 'DINT' THEN
	GetDataTypeFromPVOID := 'DINT';
	RETURN;
END_IF

IF JsonRW_DataType.GetDatatypeNameByAddress(SIZEOF(UDINT), pData) = 'UDINT' THEN
	GetDataTypeFromPVOID := 'UDINT';
	RETURN;
END_IF

IF JsonRW_DataType.GetDatatypeNameByAddress(SIZEOF(REAL), pData) = 'REAL' THEN
	GetDataTypeFromPVOID := 'REAL';
	RETURN;
END_IF

IF JsonRW_DataType.GetDatatypeNameByAddress(SIZEOF(LREAL), pData) = 'LREAL' THEN
	GetDataTypeFromPVOID := 'LREAL';
	RETURN;
END_IF

IF JsonRW_DataType.GetDatatypeNameByAddress(SIZEOF(T_MaxString), pData) = 'Tc2_System.T_MaxString' THEN
	GetDataTypeFromPVOID := 'STRING';
	RETURN;
END_IF

FOR i := 1 TO 256 DO
	IF JsonRW_DataType.GetDatatypeNameByAddress(i, pData) <> '' THEN
		GetDataTypeFromPVOID := 'STRING';
		RETURN;
	END_IF
END_FOR
END_METHOD

// Initializes event function blocks using this components's name
METHOD PROTECTED CreateEvents

// This method is called by Initialize() as required
SUPER^.CreateEvents();
F_CreateAllEventsInClass(Alarms		:= JsonFileHandlerAlarms,
						 ClassSize	:= SIZEOF(TC_EVENTS.JsonFileHandler),
						 pInitEvent := ADR(TC_EVENTS.JsonFileHandler.InitReferenceEvent),
						 Prefix		:= _Name);
END_METHOD

// Provides basic error detection and event handling for this component
METHOD PROTECTED Monitoring

// This method is called cyclically by CyclicLogic()
SUPER^.Monitoring();
IF TonTimeout.Q AND (SeqSave <> 0) AND NOT JsonFileHandlerAlarms[E_JsonFileHandler.ErrorSaveFile].bRaised THEN
	SUPER^.RaiseAlarmWithStrings(JsonFileHandlerAlarms[E_JsonFileHandler.ErrorSaveFile], _Path, '');
END_IF

IF TonTimeout.Q AND (SeqLoad <> 0) AND NOT JsonFileHandlerAlarms[E_JsonFileHandler.ErrorReadFile].bRaised THEN
	SUPER^.RaiseAlarmWithStrings(JsonFileHandlerAlarms[E_JsonFileHandler.ErrorReadFile], _Path, '');
END_IF
END_METHOD

METHOD CyclicLogic
IF _Path <> '' THEN
	FileLoadOk := JsonFileMachineConfig.LoadDocumentFromFile(sFile := _Path, bExec := FileRead); // bExec is a REFERENCE TO BOOL, the LoadDocumentFromFile method will set the variable FileRead to FALSE when done 
	FileSaveOk := JsonFileMachineConfig.SaveDocumentToFile(sFile := _Path, bExec := FileSave);	 // bExec is a REFERENCE TO BOOL, the SaveDocumentFromFile method will set the variable FileSave to FALSE when done
END_IF

// Busy and Timeout Error
_Busy := SeqSave <> 0 OR SeqLoad <> 0;
TonTimeout(IN := _Busy, PT := _Timeout);
IF TonTimeout.Q THEN
	_Error	 := TRUE;
	_ErrorID := 999;
END_IF

IF FileLoadOk THEN
	LoadDone := TRUE;
END_IF

// Save Sequence
SaveFileSequence();

// Load Sequence
LoadFileSequence();

// Call Super
SUPER^.CyclicLogic();
_CurrentAlarmSeverity := F_GetMaxSeverityRaised(Alarms := JsonFileHandlerAlarms, CurrentSeverity := _CurrentAlarmSeverity);
END_METHOD

METHOD ClearDocument
VAR_INPUT
END_VAR
JsonDoc := JsonFileMachineConfig.NewDocument();
END_METHOD

// Loads file from path, if not fould creates new file in same path
METHOD LoadFile : BOOL
LoadFile := FALSE;
IF _Path = '' THEN
	_Error	 := TRUE;
	_ErrorID := 1;
	TRACE('File Path not set!');
	RETURN;
END_IF

IF _Busy THEN
	RETURN;
END_IF

FileRead := TRUE;
SeqLoad	 := 10;
LoadFile := LoadDone;
END_METHOD

METHOD ReadAny : BOOL
VAR_INPUT
	pData : pvoid; // address of symbol
END_VAR

VAR
	pBOOL		 : POINTER TO BOOL;
	pDINT		 : POINTER TO DINT;
	pSTRING		 : POINTER TO T_MaxString;
	pLREAL		 : POINTER TO LREAL;
	PropertyName : T_MaxString;
	hrErrorCode	 : HRESULT;
	nData		 : UDINT;
	dataType	 : STRING;
	bValue		 : BOOL;
	diValue		 : DINT;
	strValue	 : T_MaxString;
	lrValue		 : LREAL;
END_VAR
ReadAny := FALSE;
IF JsonDoc = 0 OR _Busy THEN
	TRACE('File not Loaded!');
	RETURN;
END_IF

IF _Busy THEN
	RETURN;
END_IF

// Convert Variable to String
nData	 := SIZEOF(pData);
dataType := GetDataTypeFromPVOID(pData);

// BOOL
IF dataType = 'BOOL' THEN
	pBOOL		:= pData;
	nData		:= SIZEOF(pBOOL^);
	hrErrorCode := JsonRW_DataType.CopySymbolNameByAddress(nData,
														   pBOOL,
														   PropertyName,
														   SIZEOF(PropertyName));

	IF PropertyName = '' THEN
		RETURN;
	ELSE
		PropertyName := strHelp.GetName(PropertyName);
	END_IF

	ReadBOOL(PropertyName, Value => bValue);
	pBOOL^ := bValue;
END_IF

// DINT
IF dataType = 'DINT' THEN
	pDINT		:= pData;
	nData		:= SIZEOF(pDINT^);
	hrErrorCode := JsonRW_DataType.CopySymbolNameByAddress(nData,
														   pDINT,
														   PropertyName,
														   SIZEOF(PropertyName));

	IF PropertyName = '' THEN
		RETURN;
	ELSE
		PropertyName := strHelp.GetName(PropertyName);
	END_IF

	ReadDINT(PropertyName, Value => diValue);
	pDINT^ := diValue;
END_IF

// STRING 80 or 255
IF dataType = 'STRING' THEN
	pSTRING		:= pData;
	nData		:= SIZEOF(pSTRING^);
	hrErrorCode := JsonRW_DataType.CopySymbolNameByAddress(nData,
														   pSTRING,
														   PropertyName,
														   SIZEOF(PropertyName));

	IF PropertyName = '' THEN
		RETURN;
	ELSE
		PropertyName := strHelp.GetName(PropertyName);
	END_IF

	ReadSTRING(PropertyName, Value => strValue);
	pSTRING^ := strValue;
END_IF

// LREAL
IF dataType = 'LREAL' THEN
	pLREAL		:= pData;
	nData		:= SIZEOF(pLREAL^);
	hrErrorCode := JsonRW_DataType.CopySymbolNameByAddress(nData,
														   pLREAL,
														   PropertyName,
														   SIZEOF(PropertyName));

	IF PropertyName = '' THEN
		RETURN;
	ELSE
		PropertyName := strHelp.GetName(PropertyName);
	END_IF

	ReadLREAL(PropertyName, Value => lrValue);
	pLREAL^ := lrValue;
END_IF

ReadAny	 := TRUE;
JsonProp := 0;
END_METHOD

// Returns TRUE if Value has been read successfully
METHOD ReadBool : BOOL
VAR_INPUT
	PropertyName : T_MaxString;
END_VAR

VAR_OUTPUT
	Value : BOOL;
END_VAR
ReadBOOL := FALSE;
IF JsonDoc = 0 THEN
	TRACE('Document File not loaded!');
	RETURN;
END_IF

IF _Busy THEN
	RETURN;
END_IF

JsonProp := JsonFileMachineConfig.FindMember(JsonDoc, PropertyName);
Value	 := JsonFileMachineConfig.GetBOOL(JsonProp);
IF JsonProp <> 0 THEN
	ReadBOOL := TRUE;
ELSE
	ReadBOOL := THIS^.UpdateBool(PropertyName := PropertyName, Value := Value);
END_IF
END_METHOD

// Returns TRUE if Value has been read successfully
METHOD ReadDInt : BOOL
VAR_INPUT
	PropertyName : T_MaxString;
END_VAR

VAR_OUTPUT
	Value : DINT;
END_VAR
ReadDInt := FALSE;
IF JsonDoc = 0 THEN
	TRACE('Document File not loaded!');
	RETURN;
END_IF

IF _Busy THEN
	RETURN;
END_IF

JsonProp := JsonFileMachineConfig.FindMember(JsonDoc, PropertyName);
Value	 := JsonFileMachineConfig.GetInt(JsonProp);
IF JsonProp <> 0 THEN
	ReadDInt := TRUE;
ELSE
	ReadDInt := THIS^.UpdateDINT(PropertyName := PropertyName, Value := Value);
END_IF
END_METHOD

// Returns TRUE if Value has been read successfully
METHOD ReadLREAL : BOOL
VAR_INPUT
	PropertyName : T_MaxString;
END_VAR

VAR_OUTPUT
	Value : LREAL;
END_VAR
ReadLREAL := FALSE;
IF JsonDoc = 0 THEN
	TRACE('Document File not loaded!');
	RETURN;
END_IF

IF _Busy THEN
	RETURN;
END_IF

JsonProp := JsonFileMachineConfig.FindMember(JsonDoc, PropertyName);
Value	 := JsonFileMachineConfig.GetDouble(JsonProp);
IF JsonProp <> 0 THEN
	ReadLREAL := TRUE;
ELSE
	ReadLREAL := THIS^.UpdateLREAL(PropertyName := PropertyName, Value := Value);
END_IF
END_METHOD

// Returns TRUE if Value has been read successfully
METHOD ReadString : BOOL
VAR_INPUT
	PropertyName : T_MaxString;
END_VAR

VAR_OUTPUT
	Value : T_MaxString;
END_VAR
ReadString := FALSE;
IF JsonDoc = 0 THEN
	TRACE('Document File not loaded!');
	RETURN;
END_IF

IF _Busy THEN
	RETURN;
END_IF

JsonProp := JsonFileMachineConfig.FindMember(JsonDoc, PropertyName);
Value	 := JsonFileMachineConfig.GetString(JsonProp);
IF JsonProp <> 0 THEN
	ReadString := TRUE;
ELSE
	ReadString := THIS^.UpdateString(PropertyName := PropertyName, Value := Value);
END_IF
END_METHOD

METHOD ReadSymbol : BOOL
VAR_INPUT
	Datatype	 : T_MaxString;
	PropertyName : T_MaxString;
	nData		 : UDINT;
	pData		 : PVOID;
END_VAR
IF JsonDoc = 0 THEN
	TRACE('Document File not loaded!');
	RETURN;
END_IF

IF _Busy THEN
	RETURN;
END_IF

JsonProp := JsonFileMachineConfig.FindMember(JsonDoc, PropertyName);
JsonFileMachineConfig.CopyJson(v := JsonProp, pDoc := ValueJson, nDoc := SIZEOF(ValueJson));
IF JsonProp <> 0 THEN
	JsonReadWriteDataType.SetSymbolFromJson(sJson		:= ValueJson,
											sDataType	:= Datatype,
											nData		:= nData,
											pData		:= pData,
											hrErrorCode => hr);

	ReadSymbol := TRUE;
ELSE
	ReadSymbol := THIS^.UpdateSymbol(Datatype	  := Datatype,
									 PropertyName := PropertyName,
									 nData		  := nData,
									 pData		  := pData);
END_IF
END_METHOD

METHOD Reset : BOOL
SUPER^.Reset();
F_ClearAllEventsInClass(JsonFileHandlerAlarms);
_Error		  := FALSE;
_ErrorId	  := 0;
SeqSave		  := 0;
SeqLoad		  := 0;
TonTimeout.IN := FALSE;
END_METHOD

METHOD UpdateAny : BOOL
VAR_INPUT
	pData : pvoid; // address of symbol
END_VAR

VAR
	pBOOL		 : POINTER TO BOOL;
	pDINT		 : POINTER TO DINT;
	pSTRING		 : POINTER TO T_MaxString;
	pLREAL		 : POINTER TO LREAL;
	PropertyName : T_MaxString;
	hrErrorCode	 : HRESULT;
	nData		 : UDINT;
	dataType	 : STRING;
END_VAR
UpdateAny := FALSE;
IF JsonDoc = 0 OR _Busy THEN
	TRACE('File not Loaded!');
	RETURN;
END_IF

IF _Busy THEN
	RETURN;
END_IF

// Convert Variable to String
nData	 := SIZEOF(pData);
dataType := GetDataTypeFromPVOID(pData);

// BOOL
IF dataType = 'BOOL' THEN
	pBOOL		:= pData;
	nData		:= SIZEOF(pBOOL^);
	hrErrorCode := JsonRW_DataType.CopySymbolNameByAddress(nData,
														   pBOOL,
														   PropertyName,
														   SIZEOF(PropertyName));

	IF PropertyName = '' THEN
		RETURN;
	ELSE
		PropertyName := strHelp.GetName(PropertyName);
	END_IF

	UpdateBOOL(PropertyName, pBOOL^);
END_IF

// DINT
IF dataType = 'DINT' THEN
	pDINT		:= pData;
	nData		:= SIZEOF(pDINT^);
	hrErrorCode := JsonRW_DataType.CopySymbolNameByAddress(nData,
														   pDINT,
														   PropertyName,
														   SIZEOF(PropertyName));

	IF PropertyName = '' THEN
		RETURN;
	ELSE
		PropertyName := strHelp.GetName(PropertyName);
	END_IF

	UpdateDINT(PropertyName, pDINT^);
END_IF

// STRING 80 or 255
IF dataType = 'STRING' THEN
	pSTRING		:= pData;
	nData		:= SIZEOF(pSTRING^);
	hrErrorCode := JsonRW_DataType.CopySymbolNameByAddress(nData,
														   pSTRING,
														   PropertyName,
														   SIZEOF(PropertyName));

	IF PropertyName = '' THEN
		RETURN;
	ELSE
		PropertyName := strHelp.GetName(PropertyName);
	END_IF

	UpdateSTRING(PropertyName, pSTRING^);
END_IF

// LREAL
IF dataType = 'LREAL' THEN
	pLREAL		:= pData;
	nData		:= SIZEOF(pLREAL^);
	hrErrorCode := JsonRW_DataType.CopySymbolNameByAddress(nData,
														   pLREAL,
														   PropertyName,
														   SIZEOF(PropertyName));

	IF PropertyName = '' THEN
		RETURN;
	ELSE
		PropertyName := strHelp.GetName(PropertyName);
	END_IF

	UpdateLREAL(PropertyName, pLreal^);
END_IF

// Save the update to file
FileSave := TRUE;
SeqSave	 := 10;

// cleanup
UpdateAny := TRUE;
JsonProp  := 0;
END_METHOD

// Updates Json poperty, adds poperty if it does not exist
METHOD UpdateBool : BOOL
VAR_INPUT
	PropertyName : T_MaxString;
	Value		 : BOOL;
END_VAR
UpdateBool := FALSE;
IF JsonDoc = 0 OR _Busy THEN
	TRACE('File not Loaded!');
	RETURN;
END_IF

IF _Busy THEN
	RETURN;
END_IF

// Attempt to find Member
jsonProp := JsonFileMachineConfig.FindMember(JsonDoc, PropertyName);
IF JsonProp <> 0 THEN
	JsonFileMachineConfig.SetBool(JsonProp, Value);
ELSE
	JsonFileMachineConfig.AddBoolMember(JsonDoc, PropertyName, Value);
END_IF

// Save the update to file
FileSave := TRUE;
SeqSave	 := 10;

// cleanup
UpdateBool := TRUE;
JsonProp   := 0;
END_METHOD

// Updates Json poperty, adds poperty if it does not exist
METHOD UpdateDInt : BOOL
VAR_INPUT
	PropertyName : T_MaxString;
	Value		 : DINT;
END_VAR
UpdateDInt := FALSE;
IF JsonDoc = 0 OR _Busy THEN
	TRACE('File not Loaded!');
	RETURN;
END_IF

IF _Busy THEN
	RETURN;
END_IF

// Attempt to find Member
jsonProp := JsonFileMachineConfig.FindMember(JsonDoc, PropertyName);
IF JsonProp <> 0 THEN
	JsonFileMachineConfig.SetInt(JsonProp, Value);
ELSE
	JsonFileMachineConfig.AddIntMember(JsonDoc, PropertyName, Value);
END_IF

// Save the update to file
FileSave := TRUE;
SeqSave	 := 10;

// cleanup
UpdateDInt := TRUE;
JsonProp   := 0;
END_METHOD

// Updates Json poperty, adds poperty if it does not exist
METHOD UpdateLREAL : BOOL
VAR_INPUT
	PropertyName : T_MaxString;
	Value		 : LREAL;
END_VAR
UpdateLREAL := FALSE;
IF JsonDoc = 0 OR _Busy THEN
	TRACE('File not Loaded!');
	RETURN;
END_IF

IF _Busy THEN
	RETURN;
END_IF

// Attempt to find Member
jsonProp := JsonFileMachineConfig.FindMember(JsonDoc, PropertyName);
IF JsonProp <> 0 THEN
	JsonFileMachineConfig.SetDouble(JsonProp, Value);
ELSE
	JsonFileMachineConfig.AddDoubleMember(JsonDoc, PropertyName, Value);
END_IF

// Save the update to file
FileSave := TRUE;
SeqSave	 := 10;

// cleanup
UpdateLREAL := TRUE;
JsonProp	:= 0;
END_METHOD

// Updates Json poperty, adds poperty if it does not exist
METHOD UpdateString : BOOL
VAR_INPUT
	PropertyName : T_MaxString;
	Value		 : T_MaxString;
END_VAR
UpdateString := FALSE;
IF JsonDoc = 0 OR _Busy THEN
	TRACE('File not Loaded!');
	RETURN;
END_IF

IF _Busy THEN
	RETURN;
END_IF

// Attempt to find Member
jsonProp := JsonFileMachineConfig.FindMember(JsonDoc, PropertyName);
IF JsonProp <> 0 THEN
	JsonFileMachineConfig.SetString(JsonProp, Value);
ELSE
	JsonFileMachineConfig.AddStringMember(JsonDoc, PropertyName, Value);
END_IF

// Save the update to file
FileSave := TRUE;
SeqSave	 := 10;

// cleanup
UpdateString := TRUE;
JsonProp	 := 0;
END_METHOD

// Limit to String(255) for symbol
METHOD UpdateSymbol : BOOL
VAR_INPUT
	Datatype	 : T_MaxString;
	PropertyName : T_MaxString;
	nData		 : UDINT;
	pData		 : PVOID;
END_VAR
IF JsonDoc = 0 OR _Busy THEN
	TRACE('File not Loaded!');
	RETURN;
END_IF

IF _Busy THEN
	RETURN;
END_IF

// Create Json
JsonReadWriteDataType.CopyJsonStringFromSymbol(sDatatype   := Datatype,
											   nData	   := nData,
											   pData	   := pData,
											   pDoc		   := ValueJson,
											   nDoc		   := SIZEOF(ValueJson),
											   hrErrorCode => hr);

// Attempt to find Member
jsonProp := JsonFileMachineConfig.FindMember(JsonDoc, PropertyName);
IF JsonProp <> 0 THEN
	JsonFileMachineConfig.SetJson(JsonProp, ValueJson);
ELSE
	JsonFileMachineConfig.AddJsonMember(JsonDoc, PropertyName, ValueJson);
END_IF

// Save the update to file
FileSave := TRUE;
SeqSave	 := 10;

// cleanup
UpdateSymbol := TRUE;
JsonProp	 := 0;
END_METHOD

METHOD PROTECTED LoadFileSequence
VAR_INPUT
END_VAR

VAR_INST
	dirPath	 : T_MaxString;
	tryAgain : BOOL;
END_VAR

VAR
	msg : STRING;
END_VAR
CASE SeqLoad OF
	0:										// Attempt to Load File -> Command started in LoadFile()
	10:										// Load File Done
		IF NOT FileRead AND FileLoadOK THEN // File Found
			JsonDoc := JsonFileMachineConfig.GetDocumentRoot();
			SeqLoad := 0;
		END_IF

		IF NOT FileRead AND NOT FileLoadOK THEN // File not Found
			tryAgain := FALSE;
			SeqLoad	 := 20;
		END_IF

	20:									(*File Not Found - Create Directory if not exists*) ;
		fbCreateDir(bExecute := FALSE); //Prepare for rising edge in next step
		IF NOT tryAgain THEN
			dirPath := strHelp.GetPath(_Path);
		ELSE
			dirPath := strHelp.GetPath(dirPath);
		END_IF

		SeqLoad := 30;

	30:
		fbCreateDir(sNetId	  := '',
					sPathName := dirPath,
					ePath	  := PATH_GENERIC,
					bExecute  := TRUE);

		IF NOT fbCreateDir.bBusy THEN
			IF NOT fbCreateDir.bError THEN
				IF NOT tryAgain THEN
					SeqLoad := 40;
				ELSE
					tryAgain := FALSE;
					SeqLoad	 := 20;
				END_IF
			ELSE
				IF fbCreateDir.nErrId = 1827 OR fbCreateDir.nErrId = 1807 THEN
					// 0x723 Folder is already existing or invalid sPathName or ePath parameter.
					msg := CONCAT(_Path, ' File not found, but folder is existing. File will be created');
					Trace(msg);
					SeqLoad := 40;
				ELSIF fbCreateDir.nErrId = 1804 THEN
					// 0x70C Folder not found.
					msg := CONCAT('Folder is not found: ', dirPath);
					msg := CONCAT(msg, ' Reducing Path and trying again.');
					Trace(msg);
					tryagain := TRUE;
					SeqLoad	 := 20;
				ELSE
					msg := CONCAT('Create Directory Error: ', UDINT_TO_STRING(fbCreateDir.nErrId));
					Trace(msg);
					SeqLoad := 999;
				END_IF
			END_IF
		END_IF

	40: // File not found -> Create file
		JsonDoc	 := JsonFileMachineConfig.NewDocument();
		FileSave := TRUE;
		SeqLoad	 := 50;

	50: // New Document Saved
		IF NOT FileSave AND FileSaveOk THEN
			SeqLoad := 0;
		END_IF
END_CASE
END_METHOD

METHOD SaveFileSequence
VAR_INPUT
END_VAR
CASE SeqSave OF
	0:	// Attempt to save File -> Command started in UpdateXYZ()
	10: // New Document Saved
		IF NOT FileSave AND FileSaveOk THEN
			SeqSave := 0;
		END_IF
END_CASE
END_METHOD

PROPERTY PUBLIC Path : T_MaxString
GET
Path := _Path;
END_GET
SET
// Prevent the path from have a space at the end. Windows doesn't deal with that very well.
_Path := Path;
WHILE RIGHT(_Path, 1) = ' ' DO
	_Path := DELETE(_Path, 1, LEN(_Path));
END_WHILE
END_SET
END_PROPERTY

PROPERTY Timeout : TIME
SET
_Timeout := Timeout;
END_SET
END_PROPERTY

END_FUNCTION_BLOCK

// File Handlers/I_FileHandler
INTERFACE I_FileHandler EXTENDS I_BaseFB

METHOD ClearDocument
VAR_INPUT
END_VAR
END_METHOD

// Loads file from path, if not fould creates new file in same path
METHOD PUBLIC LoadFile : BOOL
END_METHOD

// Returns TRUE if Value has been read successfully
METHOD PUBLIC ReadBool : BOOL
VAR_INPUT
	PropertyName : T_MaxString;
END_VAR

VAR_OUTPUT
	Value : BOOL;
END_VAR
END_METHOD

// Returns TRUE if Value has been read successfully
METHOD PUBLIC ReadDInt : BOOL
VAR_INPUT
	PropertyName : T_MaxString;
END_VAR

VAR_OUTPUT
	Value : DINT;
END_VAR
END_METHOD

// Returns TRUE if Value has been read successfully
METHOD PUBLIC ReadLREAL : BOOL
VAR_INPUT
	PropertyName : T_MaxString;
END_VAR

VAR_OUTPUT
	Value : LREAL;
END_VAR
END_METHOD

// Returns TRUE if Value has been read successfully
METHOD PUBLIC ReadString : BOOL
VAR_INPUT
	PropertyName : T_MaxString;
END_VAR

VAR_OUTPUT
	Value : T_MaxString;
END_VAR
END_METHOD

METHOD ReadSymbol : BOOL
VAR_INPUT
	Datatype	 : T_MaxString;
	PropertyName : T_MaxString;
	nData		 : UDINT;
	pData		 : PVOID;
END_VAR
END_METHOD

METHOD PUBLIC Reset : BOOL
VAR_INPUT
END_VAR
END_METHOD

PROPERTY Timeout : TIME
SET
END_SET
END_PROPERTY

METHOD UpdateAny : BOOL
VAR_INPUT
	pData : pvoid; // address of symbol
END_VAR
END_METHOD

// Updates Json poperty, adds poperty if it does not exist
METHOD PUBLIC UpdateBool : BOOL
VAR_INPUT
	PropertyName : T_MaxString;
	Value		 : BOOL;
END_VAR
END_METHOD

// Updates Json poperty, adds poperty if it does not exist
METHOD PUBLIC UpdateDInt : BOOL
VAR_INPUT
	PropertyName : T_MaxString;
	Value		 : DINT;
END_VAR
END_METHOD

// Updates Json poperty, adds poperty if it does not exist
METHOD PUBLIC UpdateLREAL : BOOL
VAR_INPUT
	PropertyName : T_MaxString;
	Value		 : LREAL;
END_VAR
END_METHOD

// Updates Json poperty, adds poperty if it does not exist
METHOD PUBLIC UpdateString : BOOL
VAR_INPUT
	PropertyName : T_MaxString;
	Value		 : T_MaxString;
END_VAR
END_METHOD

// Limit to String(255) for symbol
METHOD UpdateSymbol : BOOL
VAR_INPUT
	Datatype	 : T_MaxString;
	PropertyName : T_MaxString;
	nData		 : UDINT;
	pData		 : PVOID;
END_VAR
END_METHOD

END_INTERFACE

// String Helper/FB_StringHelper
{attribute 'no_explicit_call' := 'This FB is a CLASS and must be accessed using methods or properties'}
FUNCTION_BLOCK FB_StringHelper

METHOD PROTECTED GetExtensionOrVarName : T_MaxString
VAR_INPUT
	input : T_MaxString;
END_VAR

VAR
	i		 : INT;
	charArry : ARRAY[0..255] OF STRING(1);
END_VAR
IF NOT ValidInput(input) THEN
	RETURN;
END_IF

charArry := StringToCharArray(input);

// Get Location of final delimiter '.'
FOR i := LEN(input) - 1 TO 0 BY -1 DO // Start at the end and find the last delimiter
	IF charArry[i] = '.' THEN
		GetExtensionOrVarName := RIGHT(input, LEN(input) - 1 - i);
		EXIT;
	END_IF
END_FOR
END_METHOD

METHOD PROTECTED GetFileNameFromPath : T_MaxString
VAR_INPUT
	input : T_MaxString;
END_VAR

VAR
	i			  : INT;
	searchResults : ARRAY[0..99] OF INT;
	tempPath	  : T_MaxString;
END_VAR
IF NOT ValidInput(input) THEN
	RETURN;
END_IF

tempPath := input; // Copy to temp variable for modification
FOR i := 0 TO LEN(input) - 1 DO
	searchResults[i] := FIND(tempPath, '\');
	IF searchResults[i] > 0 THEN
		tempPath := RIGHT(tempPath, LEN(tempPath) - searchResults[i]); // Remove begining up to and including the first delimiter
	ELSE
		EXIT; // No more delimiters remaining
	END_IF
END_FOR

GetFileNameFromPath := tempPath;
END_METHOD

METHOD PROTECTED GetFilePath : T_MaxString
VAR_INPUT
	input : T_MaxString;
END_VAR

VAR
	tempPath	  : T_MaxString;
	i			  : INT;
	searchResults : ARRAY[0..99] OF INT;
	location	  : INT;
END_VAR
IF NOT ValidInput(input) THEN
	RETURN;
END_IF

tempPath := input;								 // Copy to temp variable for modification
tempPath := LEFT(tempPath, (LEN(tempPath) - 1)); // Remove Last Character, on first pass this has no effect, but on subsequents passes this will remove the ending \

// Reduce String by removing each delimiter and counting number of characters removed to find last '\'
FOR i := 0 TO LEN(input) - 1 DO
	searchResults[i] := FIND(tempPath, '\');
	IF searchResults[i] > 0 THEN
		tempPath := RIGHT(tempPath, LEN(tempPath) - searchResults[i]); // Remove begining up to and including the first delimiter
	ELSE
		EXIT; // No more delimiters remaining
	END_IF
END_FOR

// Sum length of string to last delimiter
FOR i := 0 TO LEN(input) - 1 DO
	IF searchResults[i] > 0 THEN
		location := location + searchResults[i]; // Location of last delimiter
	ELSE
		EXIT;
	END_IF
END_FOR

GetFilePath := LEFT(input, location);
END_METHOD

METHOD GetName : T_MaxString
VAR_INPUT
	FullPath : T_MaxString;
END_VAR
IF NOT ValidInput(FullPath) THEN
	RETURN;
END_IF

// Find the First \ or . to determine if this is a File Path or Symbol Path
IF FIND(FullPath, '\') > 0 THEN
	GetName := GetFileNameFromPath(FullPath);
ELSE // symbolPath
	GetName := GetExtensionOrVarName(FullPath);
END_IF
END_METHOD

METHOD GetPath : T_MaxString
VAR_INPUT
	FullPath : T_MaxString;
END_VAR

VAR
	tempPath : T_MaxString;
END_VAR
IF NOT ValidInput(FullPath) THEN
	RETURN;
END_IF

// Find the First \ or . to determine if this is a File Path or Symbol Path
IF FIND(FullPath, '\') > 0 THEN
	GetPath := GetFilePath(FullPath);
ELSE //symbolPath
	GetPath := GetSymbolPath(FullPath);
END_IF
END_METHOD

METHOD PROTECTED GetSymbolPath : T_MaxString
VAR_INPUT
	input : T_MaxString;
END_VAR

VAR
	i		 : INT;
	charArry : ARRAY[0..255] OF STRING(1);
	tempPath : T_MaxString;
END_VAR
IF NOT ValidInput(input) THEN
	RETURN;
END_IF

charArry := StringToCharArray(input);
tempPath := input;					  // Copy to temp variable for modification
FOR i := LEN(input) - 1 TO 0 BY -1 DO // Start at the end and find the last delimiter
	IF charArry[i] = '.' THEN
		tempPath := LEFT(tempPath, i);
		EXIT;
	END_IF
END_FOR

GetSymbolPath := tempPath;
END_METHOD

METHOD PROTECTED RemoveFirstChar : T_MaxString
VAR_INPUT
	input : T_MaxString;
END_VAR
RemoveFirstChar := DELETE(input, 1, 1);
END_METHOD

METHOD PROTECTED RemoveLastChar : T_MaxString
VAR_INPUT
	input : T_MaxString;
END_VAR
RemoveLastChar := DELETE(input, 1, len(input));
END_METHOD

METHOD PROTECTED StringToCharArray : ARRAY[0..255] OF STRING(1)
VAR_INPUT
	input : T_MaxString;
END_VAR

VAR
	i		 : INT;
	end		 : INT;
	tempPath : T_MaxString;
END_VAR
IF NOT ValidInput(input) THEN
	RETURN;
END_IF

tempPath := input;

// Convert String to CharArray
FOR i := 0 TO LEN(input) - 1 DO
	StringToCharArray[i] := Left(tempPath, 1); // Return the first/next character
	tempPath			 := RemoveFirstChar(tempPath);
END_FOR
END_METHOD

METHOD PROTECTED ValidInput : BOOL
VAR_INPUT
	input : T_MaxString;
END_VAR
IF LEN(input) > 0 THEN
	ValidInput := TRUE;
ELSE
	ValidInput := FALSE;
END_IF
END_METHOD

END_FUNCTION_BLOCK

// Helper/F_CompareLREAL
FUNCTION F_CompareLREAL : BOOL
VAR_INPUT
	Val1	  : LREAL;
	Val2	  : LREAL;
	Tolerance : LREAL;
END_VAR

F_CompareLREAL := ABS(Val1 - Val2) < Tolerance;

END_FUNCTION

// Helper/F_CompareREAL
FUNCTION F_CompareREAL : BOOL
VAR_INPUT
	Val1	  : REAL;
	Val2	  : REAL;
	Tolerance : REAL;
END_VAR

F_CompareREAL := ABS(Val1 - Val2) < Tolerance;

END_FUNCTION

// Helper/F_LREAL_RoundToPlace
// Rounds an LREAL to a given number of decimal places
FUNCTION F_LREAL_RoundToPlace : LREAL // Rounded number
VAR_INPUT
	In			  : LREAL; // Number to be rounded
	DecimalPlaces : DINT;  // Number of decimal places
END_VAR

VAR
END_VAR

F_LREAL_RoundToPlace := DINT_TO_LREAL(LREAL_TO_DINT(In * (DecimalPlaces * 10))) / (DecimalPlaces * 10);

END_FUNCTION

// Helper/FB_SimpleRateLimiter
FUNCTION_BLOCK FB_SimpleRateLimiter
VAR_INPUT
	Enable		  : BOOL;
	TargetValue	  : LREAL;
	Minimum		  : LREAL;
	Maximum		  : LREAL;
	Rate_Increase : LREAL; // Units per second
	Rate_Decrease : LREAL; // Units per second
END_VAR

VAR_OUTPUT
	Y : LREAL;
END_VAR

VAR
	CycleTime_Seconds	 : LREAL;
	IncreaseRatePerCycle : LREAL;
	DecreaseRatePerCycle : LREAL;
END_VAR

IF CycleTime_Seconds = 0 THEN
	CycleTime_Seconds := UDINT_TO_LREAL(TwinCAT_SystemInfoVarList._TaskInfo[GETCURTASKINDEXEX()].CycleTime) / 10000000.0;
END_IF

IF Enable THEN
	IncreaseRatePerCycle := Rate_Increase * CycleTime_Seconds;
	DecreaseRatePerCycle := Rate_Decrease * CycleTime_Seconds;
	IF Y <> TargetValue THEN
		IF TargetValue < Y THEN
			// Decrease output
			Y := Y - DecreaseRatePerCycle;
			IF Y < Minimum THEN
				Y := Minimum;
			END_IF
		ELSIF TargetValue > Y THEN
			// Increase output
			Y := Y + IncreaseRatePerCycle;
			IF Y > Maximum THEN
				Y := Maximum;
			END_IF
		END_IF
	END_IF
END_IF

END_FUNCTION_BLOCK

// Project Information/F_GetCompany
// This function has been automatically generated from the project information.
{attribute 'signature_flag' := '1073741824'}
{attribute 'TcGenerated'}
{attribute 'no-analysis'}
FUNCTION F_GetCompany : WSTRING
VAR_INPUT
	
END_VAR

F_GetCompany := "Beckhoff Automation LLC";

END_FUNCTION

// Project Information/F_GetTitle
// This function has been automatically generated from the project information.
{attribute 'signature_flag' := '1073741824'}
{attribute 'TcGenerated'}
{attribute 'no-analysis'}
FUNCTION F_GetTitle : WSTRING
VAR_INPUT
	
END_VAR

F_GetTitle := "SPT Utilities";

END_FUNCTION

// Project Information/F_GetVersion
// This function has been automatically generated from the project information.
{attribute 'signature_flag' := '1073741824'}
{attribute 'TcGenerated'}
{attribute 'no-analysis'}
FUNCTION F_GetVersion : ST_LibVersion
VAR_INPUT
	
END_VAR

F_GetVersion.iMajor := 4;
F_GetVersion.iMinor := 0;
F_GetVersion.iBuild := 1;
F_GetVersion.iRevision := 0;
F_GetVersion.sVersion := '4.0.1';
F_GetVersion.nFlags := 1;

END_FUNCTION

// Trace Listener/FB_MessageListener
FUNCTION_BLOCK FINAL FB_MessageListener EXTENDS FB_ListenerBase2
VAR
	Json		  : FB_JsonDomParser; // Parse JSON attribute of messages
	JsonAttribute : STRING(10000);	  // Holds JSON attribute
	hr			  : HRESULT;		  // Signals JSON attribute was successfully read
	ipListener	  : I_TraceListener;  // Receives callback once message is processed
END_VAR

PROPERTY Listener : I_TraceListener
SET
ipListener := Listener;
END_SET
END_PROPERTY

METHOD OnMessageSent : HRESULT
VAR_INPUT
	fbEvent : REFERENCE TO FB_TcEvent;
END_VAR

VAR
	Message		 : ST_TraceMessage;
	JsonDocument : SJsonValue;
	JsonProperty : SJsonValue;
END_VAR
hr := fbEvent.GetJsonAttribute(JsonAttribute, SIZEOF(JsonAttribute));
IF SUCCEEDED(hr) THEN
	JsonDocument := Json.ParseDocument(JsonAttribute);
	IF Json.HasMember(JsonDocument, 'DCTimeStamp') THEN
		JsonProperty	  := Json.FindMember(JsonDocument, 'DCTimeStamp');
		Message.Timestamp := Json.GetString(JsonProperty);
	END_IF

	IF Json.HasMember(JsonDocument, 'Instance') THEN
		JsonProperty   := Json.FindMember(JsonDocument, 'Instance');
		Message.Source := Json.GetString(JsonProperty);
	END_IF

	IF Json.HasMember(JsonDocument, 'Context') THEN
		JsonProperty	:= Json.FindMember(JsonDocument, 'Context');
		Message.Context := Json.GetString(JsonProperty);
	END_IF

	IF Json.HasMember(JsonDocument, 'ScanCount') THEN
		JsonProperty	  := Json.FindMember(JsonDocument, 'ScanCount');
		Message.ScanCount := Json.GetUint(JsonProperty);
	END_IF

	IF Json.HasMember(JsonDocument, 'Flags') THEN
		JsonProperty  := Json.FindMember(JsonDocument, 'Flags');
		Message.Flags := Json.GetUint(JsonProperty);
	END_IF

	IF Json.HasMember(JsonDocument, 'Message') THEN
		JsonProperty	:= Json.FindMember(JsonDocument, 'Message');
		Message.Message := Json.GetString(JsonProperty);
	END_IF

	IF Json.HasMember(JsonDocument, 'ExtendedInfo') THEN
		JsonProperty := Json.FindMember(JsonDocument, 'ExtendedInfo');
		Message.Json := Json.GetString(JsonProperty);
	END_IF

	IF ipListener <> 0 THEN
		// Notify listener of message data
		ipListener.OnTraceReceived(Message);
	END_IF
END_IF

OnMessageSent := S_OK; // in order to receive more callbacks (Set <> S_OK in order to cancel the callbacks for this program cycle.)
END_METHOD

END_FUNCTION_BLOCK

// Trace Listener/I_TraceListener
INTERFACE I_TraceListener

METHOD OnTraceReceived
VAR_INPUT
	Message : ST_TraceMessage;
END_VAR
END_METHOD

END_INTERFACE

// Trace Listener/FB_TraceListenerBase
FUNCTION_BLOCK ABSTRACT FB_TraceListenerBase EXTENDS FB_CyclicFB IMPLEMENTS I_TraceListener
VAR_INPUT
END_VAR

VAR_OUTPUT
END_VAR

VAR
	MessageListener : FB_MessageListener;
END_VAR

METHOD PUBLIC CyclicLogic
IF NOT _InitComplete THEN
	_InitComplete := Initialize();
	RETURN;
END_IF

MessageListener.Execute();
END_METHOD

METHOD PROTECTED Initialize : BOOL
VAR
	ListenerFilter : FB_TcEventFilter;
	hr			   : HRESULT;
END_VAR
MessageListener.Listener := THIS^;									 // For callbacks on message received
ListenerFilter.Clear().EventClass.EqualTo(TC_EVENT_CLASSES.Tracing); // Filter events by tracing class
hr := MessageListener.Subscribe2(ListenerFilter);					 // Subscribe to retrieve defined events
IF SUCCEEDED(hr) THEN
	Initialize := TRUE;
END_IF
END_METHOD

METHOD ABSTRACT OnTraceReceived
VAR_INPUT
	Message : ST_TraceMessage;
END_VAR
// Override this method to implement your specific handling
END_METHOD

END_FUNCTION_BLOCK

// Tree_IndexBased/FB_Tree_IndexBased
// Maintains a hierachical representation of a group of parent/child relationships 
FUNCTION_BLOCK FB_Tree_IndexBased IMPLEMENTS I_Tree_IndexBased
VAR_IN_OUT
	Nodes : ARRAY[0..63] OF ST_Tree_IndexBased_Node; // Holding array
END_VAR

VAR_INPUT
	Head : STRING; // Name of the root element
END_VAR

VAR
	Initialized	 : BOOL;
	NodeCount	 : DINT;
	NewNodeIndex : DINT;
	HeadIndex	 : DINT;

	//"Temp" variables for use in AddNodeAsChildByName
	ParentIndex : DINT;
	ChildCount	: DINT;
END_VAR

IF NOT Initialized THEN
	Initialize();
END_IF

// Add a child element to a node
METHOD AddNodeAsChildByName
VAR_INPUT
	NewName	   : STRING; // Name of the new element
	ParentName : STRING; // Name of the parent element
END_VAR
ParentIndex := GetIndexByName(ParentName); // Find the index value of the designated parent node
ChildCount	:= Nodes[ParentIndex].ChildCount;
IF ParentIndex >= 0 THEN										// If GetIndex was successful
	IF (Nodes[ParentIndex].ChildCount < 64) THEN				// If the parent is not at max child count
		Nodes[NewNodeIndex].Name				:= NewName;		// assign new node name to next empty node in list
		Nodes[NewNodeIndex].Parent				:= ParentIndex; // assign the parent node to the new child node
		Nodes[NewNodeIndex].Depth				:= Nodes[ParentIndex].Depth + 1;
		Nodes[ParentIndex].Children[ChildCount] := NewNodeIndex;	 // assign the new node location as the next child in the parent
		NewNodeIndex							:= NewNodeIndex + 1; // Increment to next empty node
		Nodes[ParentIndex].ChildCount			:= ChildCount + 1;
	END_IF
END_IF
END_METHOD

// Searches the current branch for a node matching the provided name and returns its index

// The index of the matching node (-1 if no match found)
METHOD PUBLIC GetIndexByName : DINT
VAR_INPUT
	Name : STRING; // Node to search for
END_VAR

VAR
	i : DINT;
END_VAR
FOR i := 0 TO NodeCount DO
	IF Nodes[i].Name = Name THEN
		GetIndexByName := i;
		RETURN;
	END_IF
END_FOR

GetIndexByName := -1;
END_METHOD

METHOD PRIVATE Initialize
NodeCount := 64;
IF NodeCount >= 0 THEN
	HeadIndex				:= 0;
	Nodes[HeadIndex].Name	:= Head;
	Nodes[HeadIndex].Depth	:= 0;
	Nodes[HeadIndex].Parent := -1;
	NewNodeIndex			:= HeadIndex + 1;
END_IF
END_METHOD

END_FUNCTION_BLOCK

// Tree_IndexBased/I_Tree_IndexBased
INTERFACE I_Tree_IndexBased

METHOD PUBLIC AddNodeAsChildByName
VAR_INPUT
	NewName	   : STRING;
	ParentName : STRING;
END_VAR
END_METHOD

END_INTERFACE
